PROGRAM main
  VAR
    At_Entry AT %IX0.0 : BOOL;
    At_Load AT %IX0.1 : BOOL;
    At_Left AT %IX0.2 : BOOL;
    At_Middle AT %IX0.3 : BOOL;
    At_Right AT %IX0.4 : BOOL;
    At_Unload AT %IX0.5 : BOOL;
    At_Exit AT %IX0.6 : BOOL;
    Moving_X AT %IX0.7 : BOOL;
    Moving_Z AT %IX1.0 : BOOL;
    Start_Button AT %IX1.1 : BOOL;
    Reset_Button AT %IX1.2 : BOOL;
    Stop_Button AT %IX1.3 : BOOL;
    Emergency_Stop AT %IX1.4 : BOOL;
    Auto_Mode AT %IX1.5 : BOOL;
    FIO_Running AT %IX1.6 : BOOL;
    Entry_Conveyor AT %QX0.0 : BOOL;
    Load_Conveyor AT %QX0.1 : BOOL;
    Forks_Left AT %QX0.2 : BOOL;
    Forks_Right AT %QX0.3 : BOOL;
    Lift AT %QX0.4 : BOOL;
    Unload_Conveyor AT %QX0.5 : BOOL;
    Exit_Conveyor AT %QX0.6 : BOOL;
    Start_Light AT %QX0.7 : BOOL;
    Reset_Light AT %QX1.0 : BOOL;
    Stop_Light AT %QX1.1 : BOOL;
    Target_Position AT %QW0 : INT;
    Init_Req : BOOL;
    Init_Cmd : BOOL;
    Boot_Done : BOOL;
    Fault_Latch : BOOL;
    System_Run : BOOL;
    Idle_Enter : BOOL;
    S0_Idle : BOOL;
    S1_Load_ForkOut : BOOL;
    S2_Load_LiftUp : BOOL;
    S3_Load_ForkIn : BOOL;
    S4_Move_To_Cell : BOOL;
    S5_Cell_ForkOut : BOOL;
    S6_Cell_LiftDown : BOOL;
    S7_Cell_ForkIn : BOOL;
    S8_Get_ForkOut : BOOL;
    S9_Get_LiftUp : BOOL;
    S10_Get_ForkIn : BOOL;
    S11_Move_To_Unload : BOOL;
    S12_Unload_ForkOut : BOOL;
    S13_Unload_LiftDown : BOOL;
    S14_Unload_ForkIn : BOOL;
    CellOut_Req : BOOL;
    Ext_Load : BOOL;
    Ext_Cell : BOOL;
    Ext_Unload : BOOL;
    Lift_Req : BOOL;
    Unload_Run : BOOL;
    T_LiftA : TON;
    T_LiftB : TON;
    T_LiftC : TON;
    T_LiftD : TON;
    T_Move1 : TON;
    T_Move2 : TON;
  END_VAR

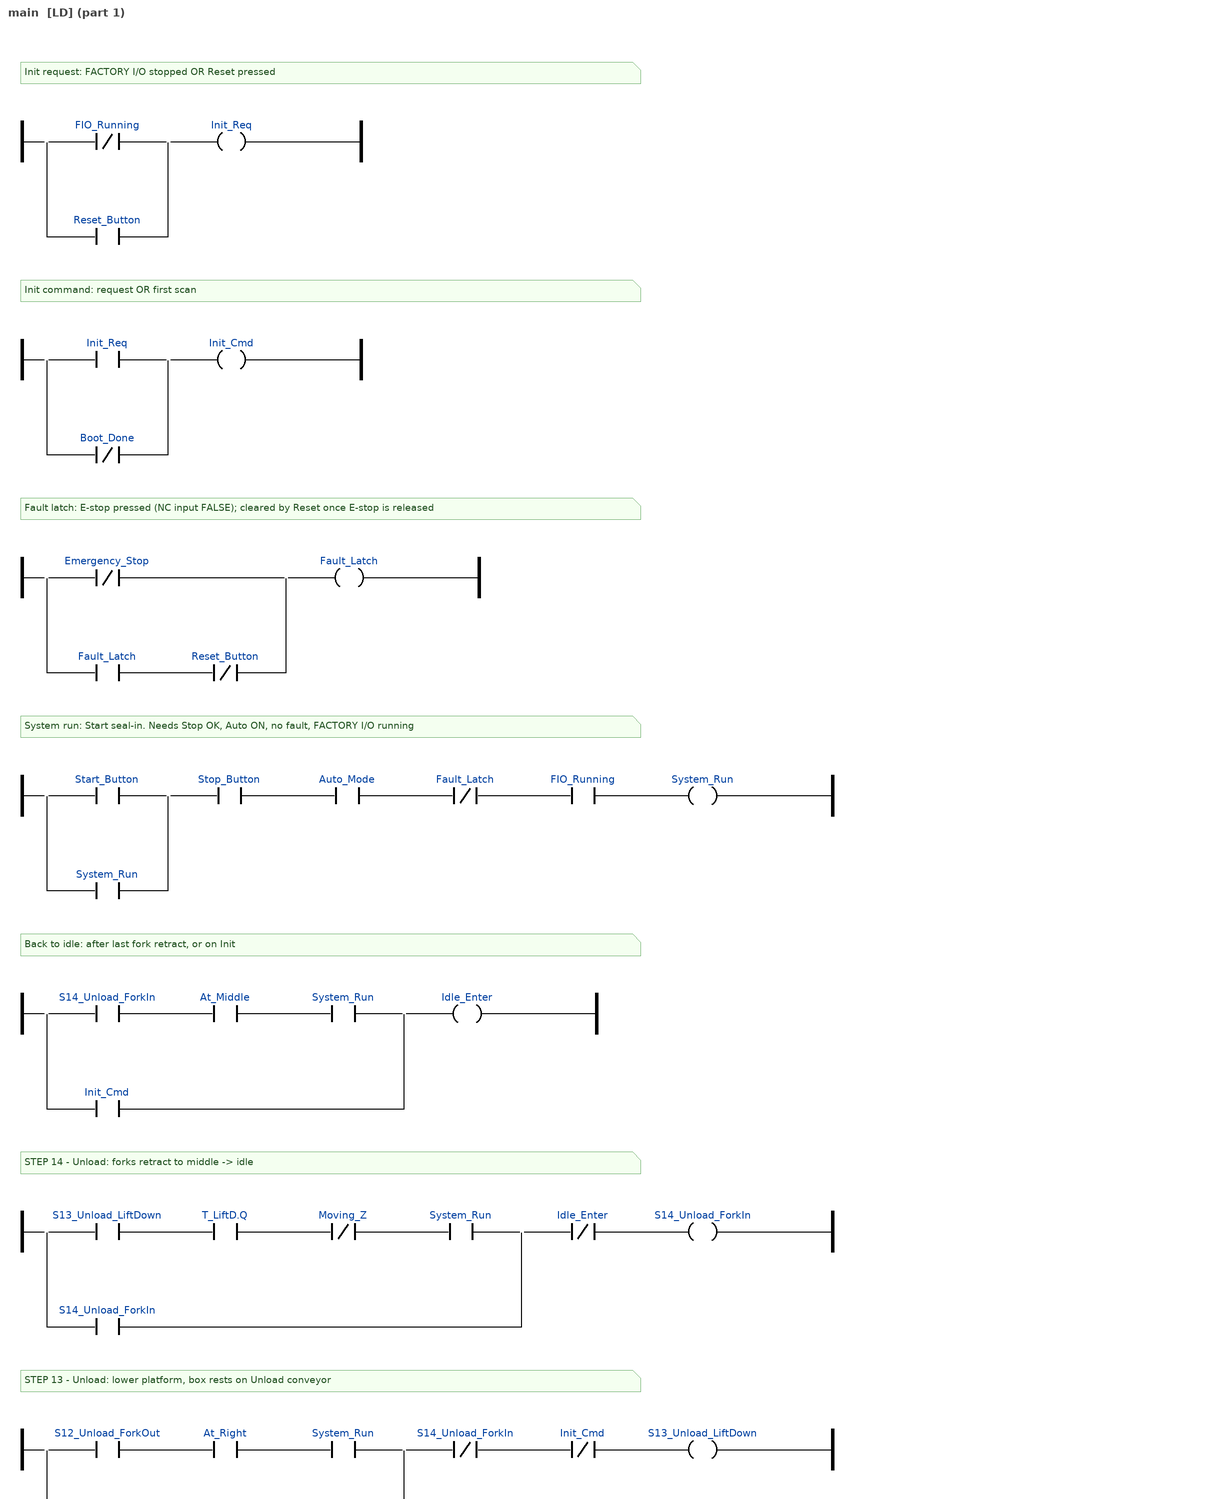
(* LD diagram, written out as Structured Text *)
(* Init request: FACTORY I/O stopped OR Reset pressed *)
Init_Req := NOT FIO_Running OR Reset_Button;
(* Init command: request OR first scan *)
Init_Cmd := Init_Req OR NOT Boot_Done;
(* Fault latch: E-stop pressed (NC input FALSE); cleared by Reset once E-stop is released *)
Fault_Latch := NOT Emergency_Stop OR Fault_Latch AND NOT Reset_Button;
(* System run: Start seal-in. Needs Stop OK, Auto ON, no fault, FACTORY I/O running *)
System_Run := (Start_Button OR System_Run) AND Stop_Button AND Auto_Mode AND NOT Fault_Latch AND FIO_Running;
(* Back to idle: after last fork retract, or on Init *)
Idle_Enter := S14_Unload_ForkIn AND At_Middle AND System_Run OR Init_Cmd;
(* STEP 14 - Unload: forks retract to middle -> idle *)
S14_Unload_ForkIn := (S13_Unload_LiftDown AND T_LiftD.Q AND NOT Moving_Z AND System_Run OR S14_Unload_ForkIn) AND NOT Idle_Enter;
(* STEP 13 - Unload: lower platform, box rests on Unload conveyor *)
S13_Unload_LiftDown := (S12_Unload_ForkOut AND At_Right AND System_Run OR S13_Unload_LiftDown) AND NOT S14_Unload_ForkIn AND NOT Init_Cmd;
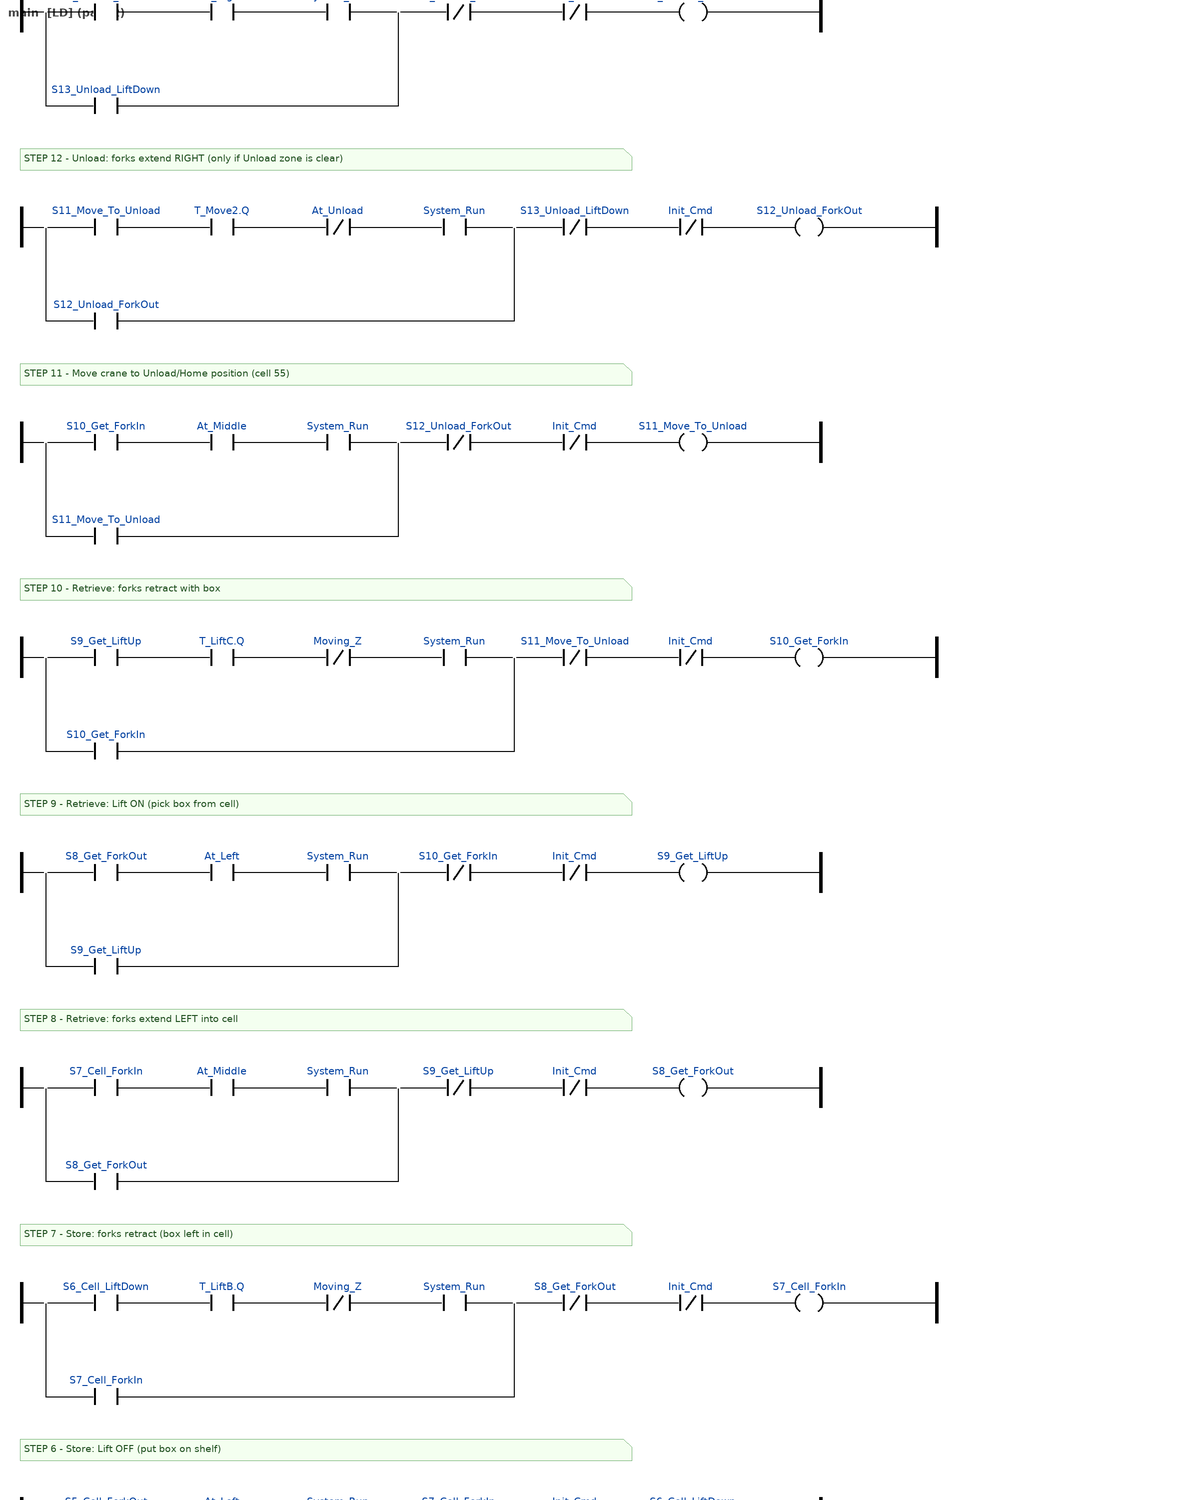
(* STEP 12 - Unload: forks extend RIGHT (only if Unload zone is clear) *)
S12_Unload_ForkOut := (S11_Move_To_Unload AND T_Move2.Q AND NOT At_Unload AND System_Run OR S12_Unload_ForkOut) AND NOT S13_Unload_LiftDown AND NOT Init_Cmd;
(* STEP 11 - Move crane to Unload/Home position (cell 55) *)
S11_Move_To_Unload := (S10_Get_ForkIn AND At_Middle AND System_Run OR S11_Move_To_Unload) AND NOT S12_Unload_ForkOut AND NOT Init_Cmd;
(* STEP 10 - Retrieve: forks retract with box *)
S10_Get_ForkIn := (S9_Get_LiftUp AND T_LiftC.Q AND NOT Moving_Z AND System_Run OR S10_Get_ForkIn) AND NOT S11_Move_To_Unload AND NOT Init_Cmd;
(* STEP 9 - Retrieve: Lift ON (pick box from cell) *)
S9_Get_LiftUp := (S8_Get_ForkOut AND At_Left AND System_Run OR S9_Get_LiftUp) AND NOT S10_Get_ForkIn AND NOT Init_Cmd;
(* STEP 8 - Retrieve: forks extend LEFT into cell *)
S8_Get_ForkOut := (S7_Cell_ForkIn AND At_Middle AND System_Run OR S8_Get_ForkOut) AND NOT S9_Get_LiftUp AND NOT Init_Cmd;
(* STEP 7 - Store: forks retract (box left in cell) *)
S7_Cell_ForkIn := (S6_Cell_LiftDown AND T_LiftB.Q AND NOT Moving_Z AND System_Run OR S7_Cell_ForkIn) AND NOT S8_Get_ForkOut AND NOT Init_Cmd;
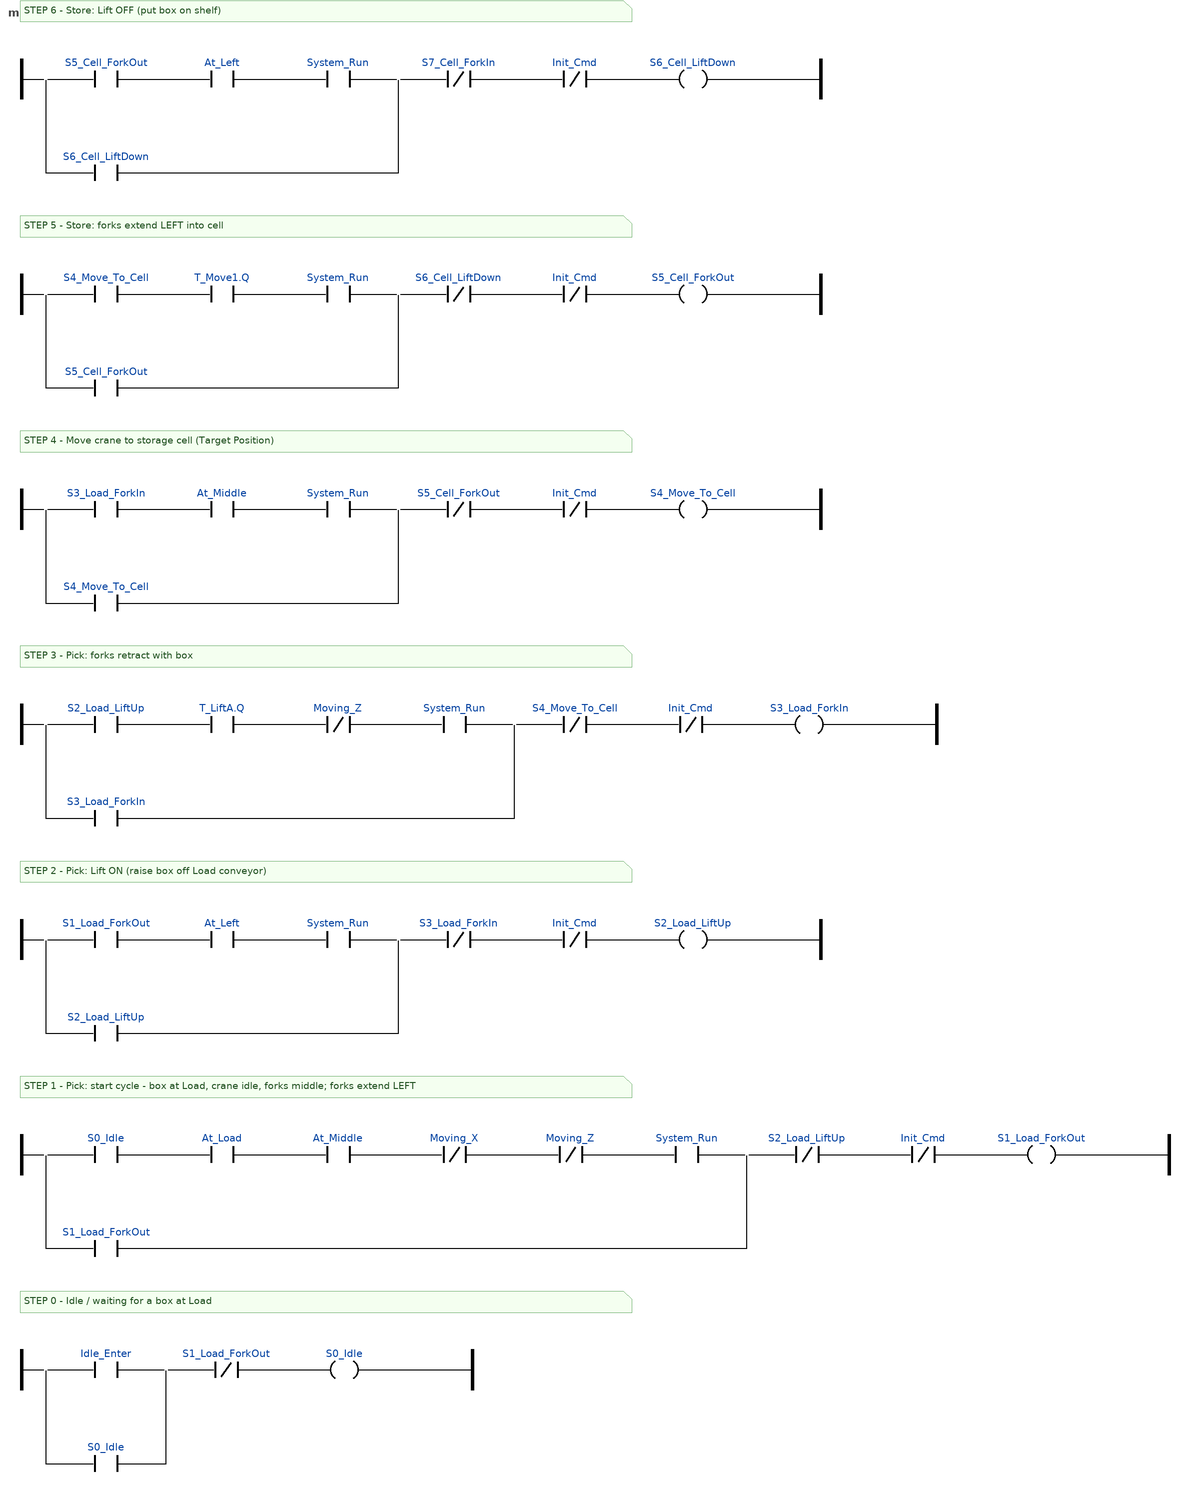
(* STEP 6 - Store: Lift OFF (put box on shelf) *)
S6_Cell_LiftDown := (S5_Cell_ForkOut AND At_Left AND System_Run OR S6_Cell_LiftDown) AND NOT S7_Cell_ForkIn AND NOT Init_Cmd;
(* STEP 5 - Store: forks extend LEFT into cell *)
S5_Cell_ForkOut := (S4_Move_To_Cell AND T_Move1.Q AND System_Run OR S5_Cell_ForkOut) AND NOT S6_Cell_LiftDown AND NOT Init_Cmd;
(* STEP 4 - Move crane to storage cell (Target Position) *)
S4_Move_To_Cell := (S3_Load_ForkIn AND At_Middle AND System_Run OR S4_Move_To_Cell) AND NOT S5_Cell_ForkOut AND NOT Init_Cmd;
(* STEP 3 - Pick: forks retract with box *)
S3_Load_ForkIn := (S2_Load_LiftUp AND T_LiftA.Q AND NOT Moving_Z AND System_Run OR S3_Load_ForkIn) AND NOT S4_Move_To_Cell AND NOT Init_Cmd;
(* STEP 2 - Pick: Lift ON (raise box off Load conveyor) *)
S2_Load_LiftUp := (S1_Load_ForkOut AND At_Left AND System_Run OR S2_Load_LiftUp) AND NOT S3_Load_ForkIn AND NOT Init_Cmd;
(* STEP 1 - Pick: start cycle - box at Load, crane idle, forks middle; forks extend LEFT *)
S1_Load_ForkOut := (S0_Idle AND At_Load AND At_Middle AND NOT Moving_X AND NOT Moving_Z AND System_Run OR S1_Load_ForkOut) AND NOT S2_Load_LiftUp AND NOT Init_Cmd;
(* STEP 0 - Idle / waiting for a box at Load *)
S0_Idle := (Idle_Enter OR S0_Idle) AND NOT S1_Load_ForkOut;
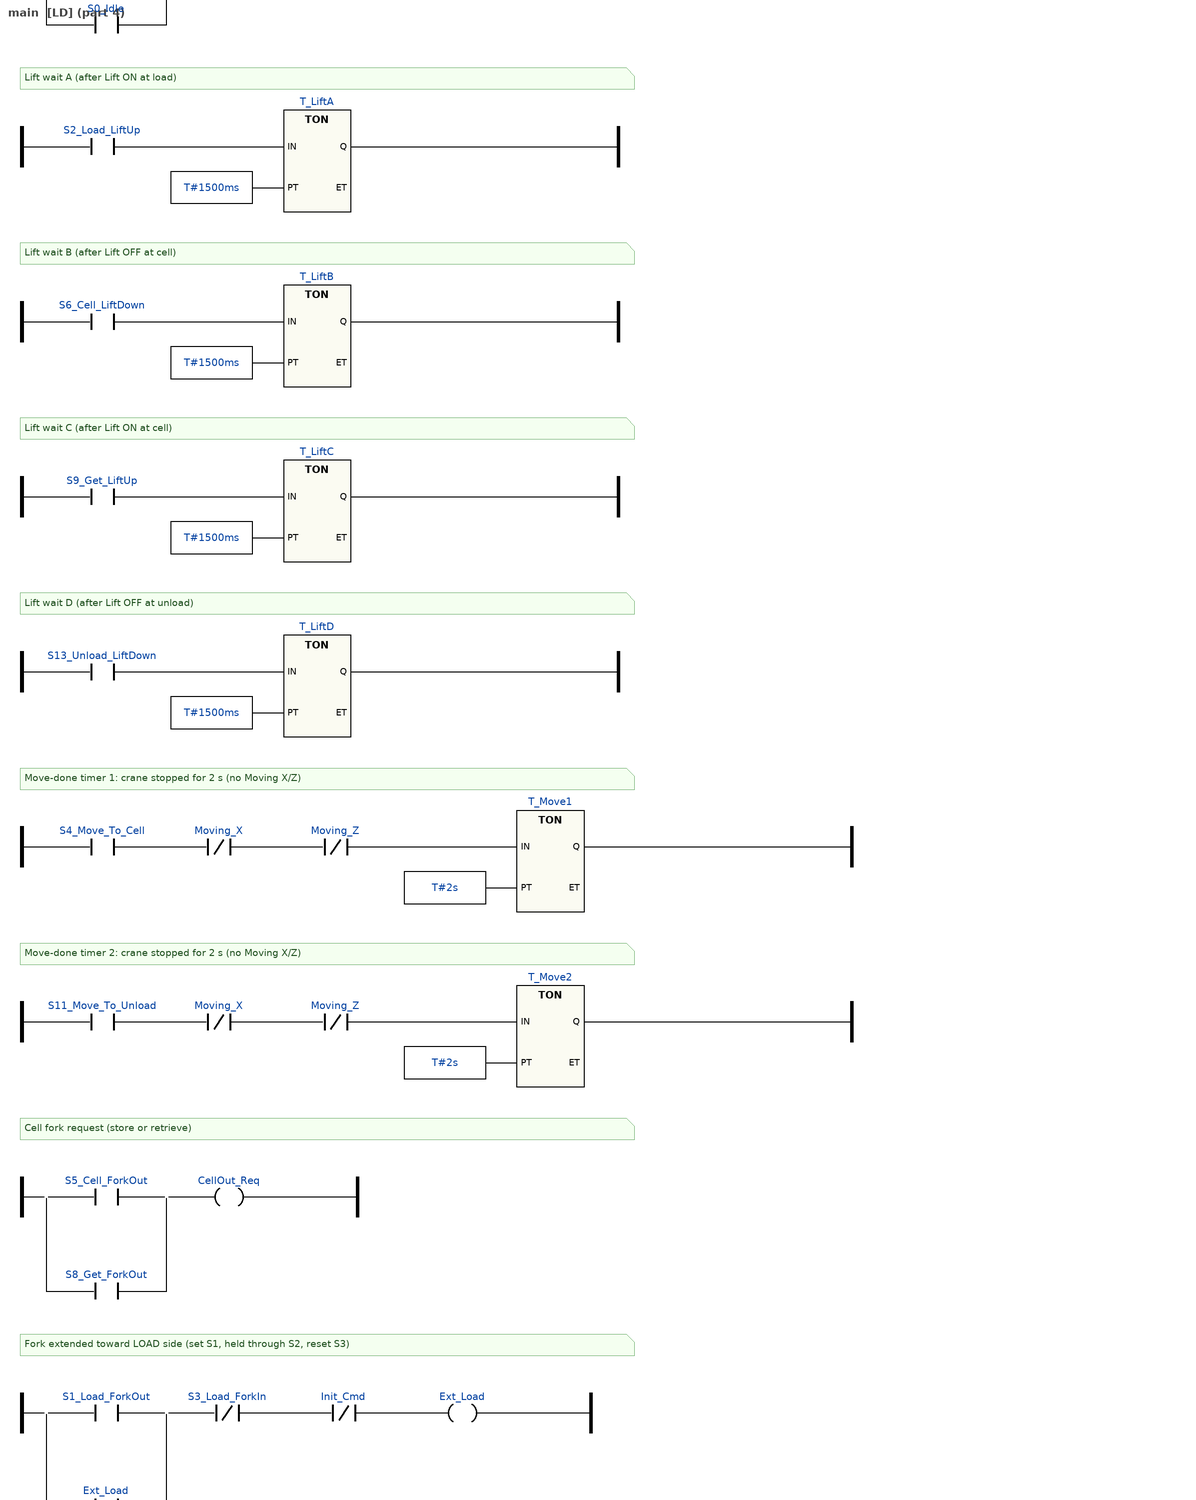
(* Lift wait A (after Lift ON at load) *)
(* Lift wait B (after Lift OFF at cell) *)
(* Lift wait C (after Lift ON at cell) *)
(* Lift wait D (after Lift OFF at unload) *)
(* Move-done timer 1: crane stopped for 2 s (no Moving X/Z) *)
(* Move-done timer 2: crane stopped for 2 s (no Moving X/Z) *)
(* Cell fork request (store or retrieve) *)
CellOut_Req := S5_Cell_ForkOut OR S8_Get_ForkOut;
(* Fork extended toward LOAD side (set S1, held through S2, reset S3) *)
Ext_Load := (S1_Load_ForkOut OR Ext_Load) AND NOT S3_Load_ForkIn AND NOT Init_Cmd;
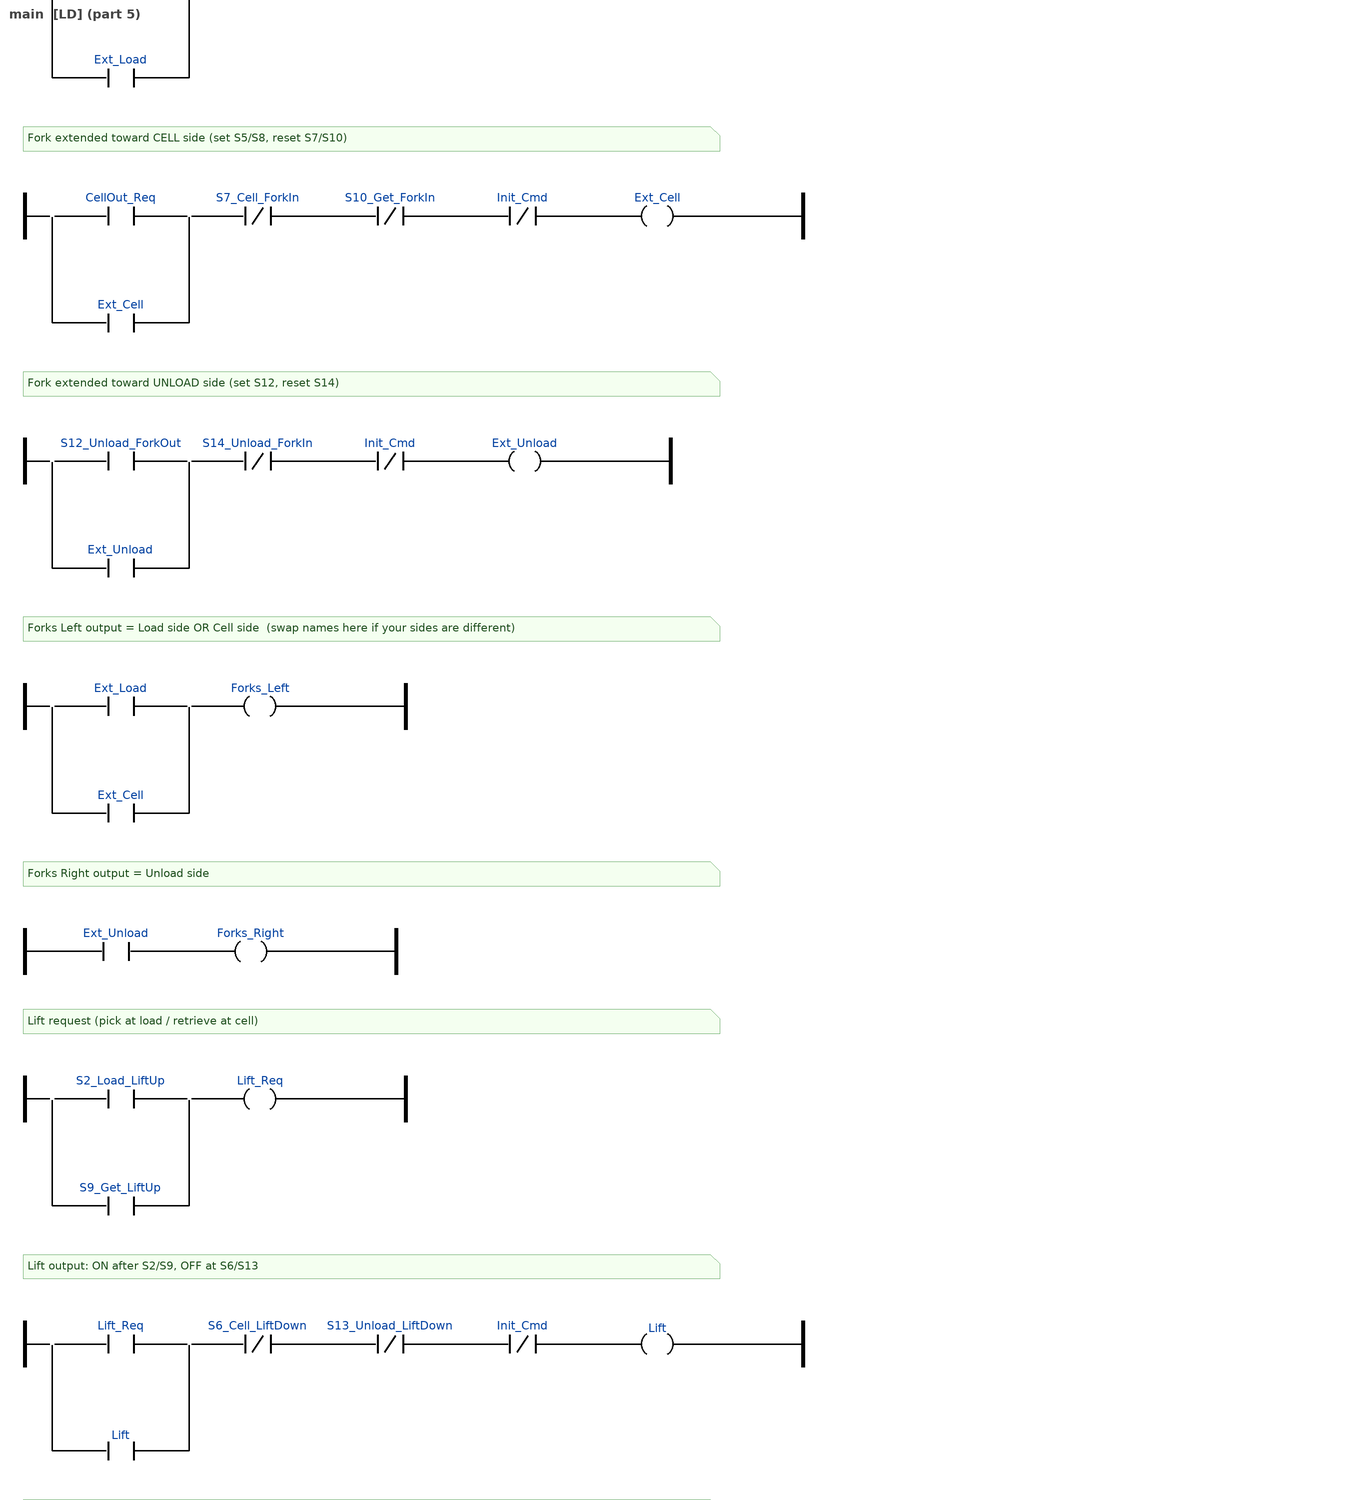
(* Fork extended toward CELL side (set S5/S8, reset S7/S10) *)
Ext_Cell := (CellOut_Req OR Ext_Cell) AND NOT S7_Cell_ForkIn AND NOT S10_Get_ForkIn AND NOT Init_Cmd;
(* Fork extended toward UNLOAD side (set S12, reset S14) *)
Ext_Unload := (S12_Unload_ForkOut OR Ext_Unload) AND NOT S14_Unload_ForkIn AND NOT Init_Cmd;
(* Forks Left output = Load side OR Cell side  (swap names here if your sides are different) *)
Forks_Left := Ext_Load OR Ext_Cell;
(* Forks Right output = Unload side *)
Forks_Right := Ext_Unload;
(* Lift request (pick at load / retrieve at cell) *)
Lift_Req := S2_Load_LiftUp OR S9_Get_LiftUp;
(* Lift output: ON after S2/S9, OFF at S6/S13 *)
Lift := (Lift_Req OR Lift) AND NOT S6_Cell_LiftDown AND NOT S13_Unload_LiftDown AND NOT Init_Cmd;
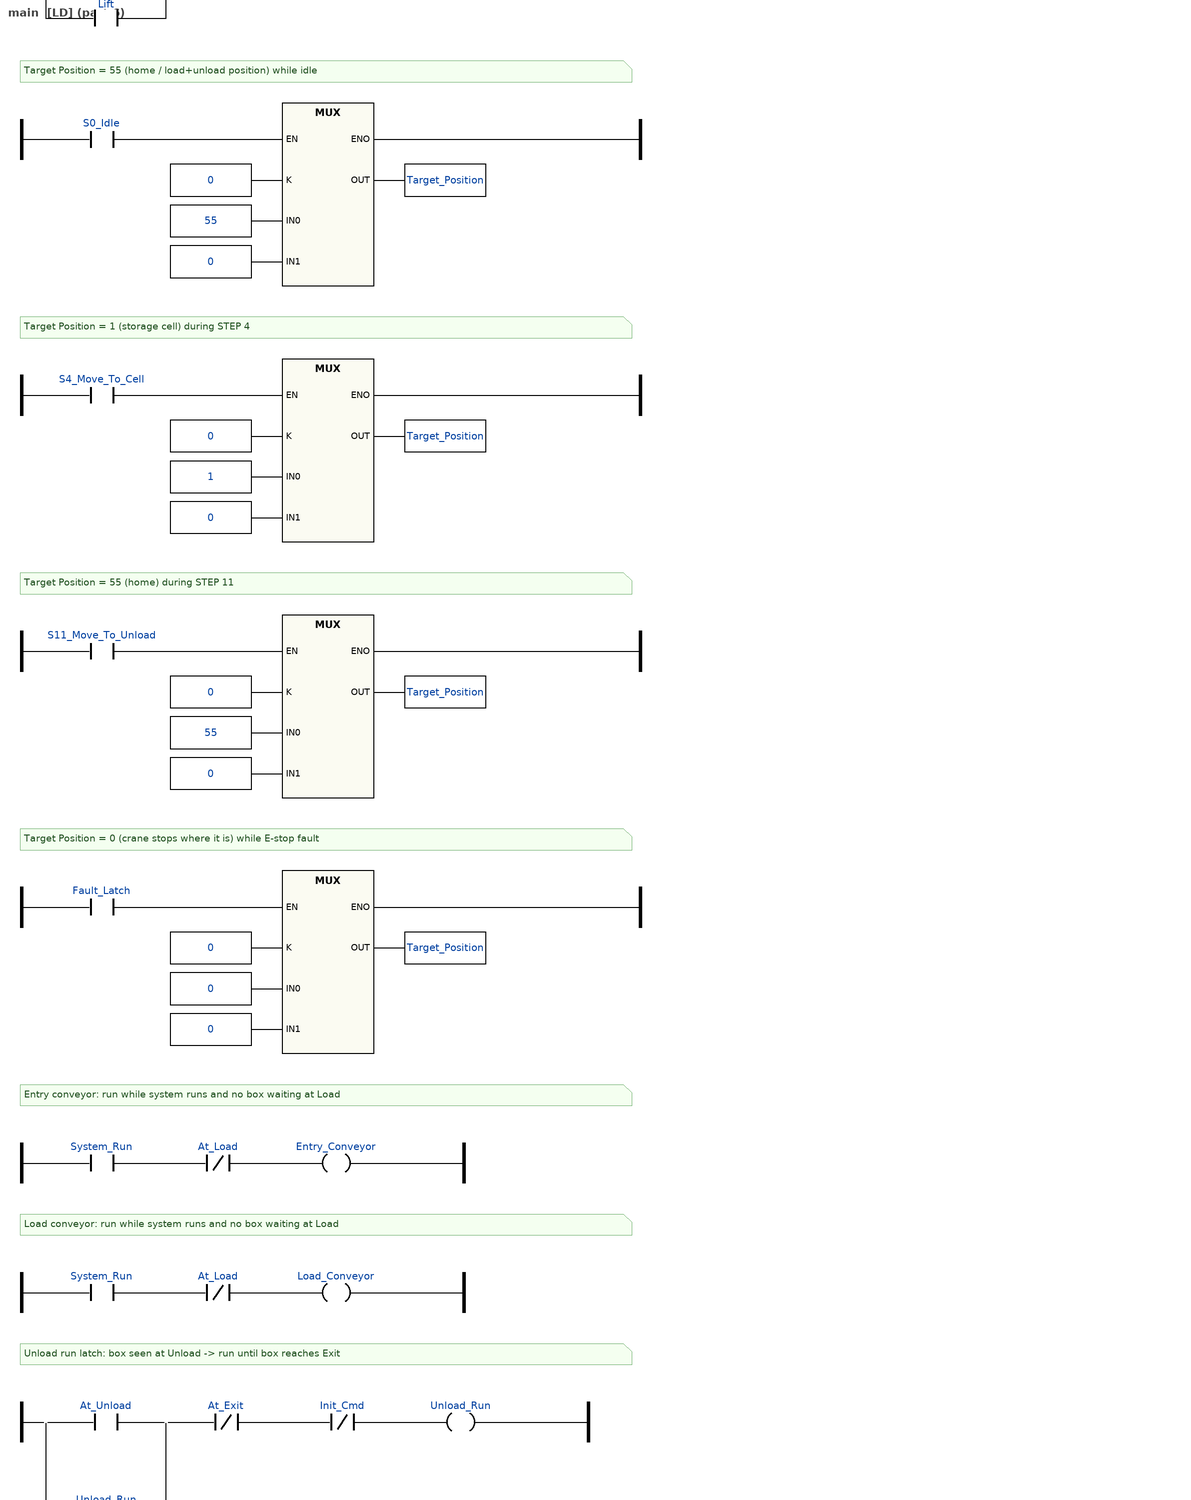
(* Target Position = 55 (home / load+unload position) while idle *)
IF S0_Idle THEN Target_Position := MUX(0, 55, 0); END_IF;
(* Target Position = 1 (storage cell) during STEP 4 *)
IF S4_Move_To_Cell THEN Target_Position := MUX(0, 1, 0); END_IF;
(* Target Position = 55 (home) during STEP 11 *)
IF S11_Move_To_Unload THEN Target_Position := MUX(0, 55, 0); END_IF;
(* Target Position = 0 (crane stops where it is) while E-stop fault *)
IF Fault_Latch THEN Target_Position := MUX(0, 0, 0); END_IF;
(* Entry conveyor: run while system runs and no box waiting at Load *)
Entry_Conveyor := System_Run AND NOT At_Load;
(* Load conveyor: run while system runs and no box waiting at Load *)
Load_Conveyor := System_Run AND NOT At_Load;
(* Unload run latch: box seen at Unload -> run until box reaches Exit *)
Unload_Run := (At_Unload OR Unload_Run) AND NOT At_Exit AND NOT Init_Cmd;
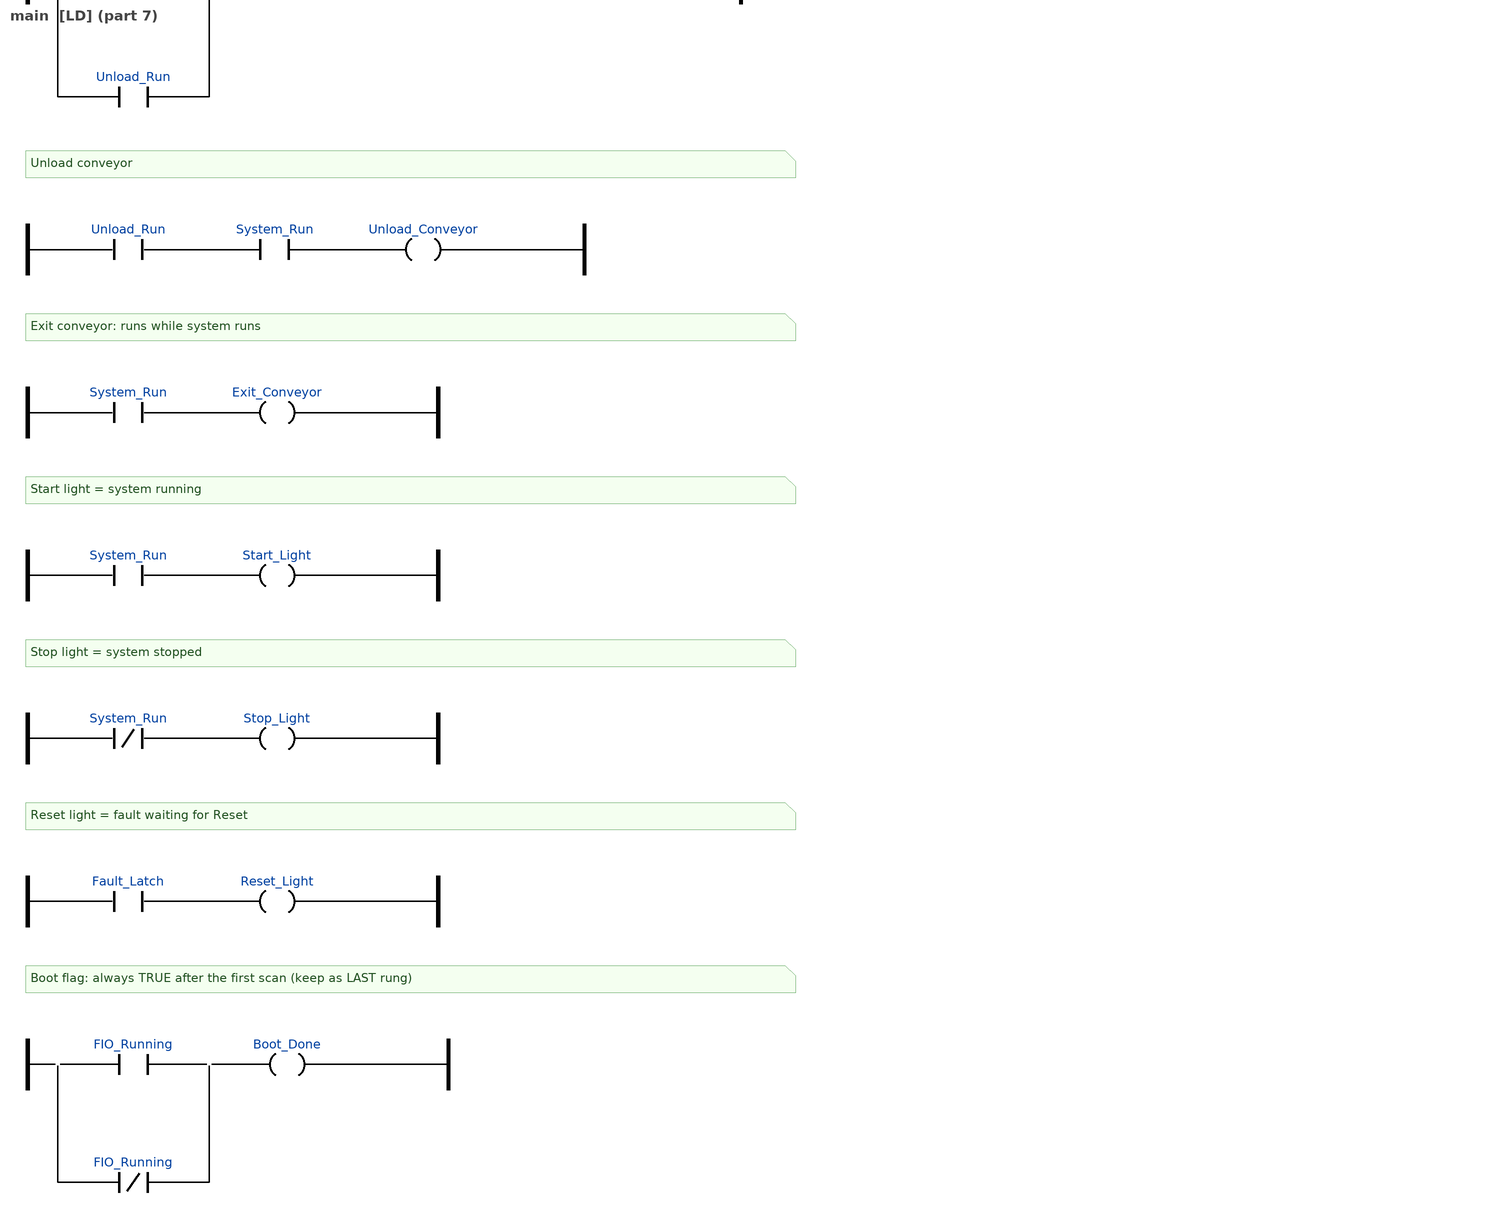
(* Unload conveyor *)
Unload_Conveyor := Unload_Run AND System_Run;
(* Exit conveyor: runs while system runs *)
Exit_Conveyor := System_Run;
(* Start light = system running *)
Start_Light := System_Run;
(* Stop light = system stopped *)
Stop_Light := NOT System_Run;
(* Reset light = fault waiting for Reset *)
Reset_Light := Fault_Latch;
(* Boot flag: always TRUE after the first scan (keep as LAST rung) *)
Boot_Done := FIO_Running OR NOT FIO_Running;
T_LiftA(IN := S2_Load_LiftUp, PT := T#1500ms);
T_LiftB(IN := S6_Cell_LiftDown, PT := T#1500ms);
T_LiftC(IN := S9_Get_LiftUp, PT := T#1500ms);
T_LiftD(IN := S13_Unload_LiftDown, PT := T#1500ms);
T_Move1(IN := S4_Move_To_Cell AND NOT Moving_X AND NOT Moving_Z, PT := T#2s);
T_Move2(IN := S11_Move_To_Unload AND NOT Moving_X AND NOT Moving_Z, PT := T#2s);
END_PROGRAM
